# EPICS autosave request: measCompApp/Db/measCompMCS_settings.req
$(P)PresetReal
$(P)Dwell
$(P)Prescale
$(P)ChannelAdvance
$(P)ReadAll.SCAN
$(P)NuseAll
$(P)EnableClientWait
